// TIA Portal V17 export
// export: Created 2023-02-14T02:49:46.84947Z, ExportSetting WithDefaults, DisplayName Totally Integrated Automation Portal, DisplayVersion V17, DisplayName TIA Portal Openness, DisplayVersion V17, DisplayName TIA Portal Teamcenter Gateway, DisplayVersion V17, DisplayName TIA Portal Version Control Interface, DisplayVersion V17, DisplayName SINAMICS Startdrive Advanced, DisplayVersion V17, DisplayName SINAMICS Startdrive G130, G150, S120, S150, SINAMICS MV, S210, DisplayVersion V17, DisplayName SINAMICS Startdrive G110M, G120, G120C, G120D, G120P, G115D, DisplayVersion V17, DisplayName STEP 7 Professional, DisplayVersion V17, DisplayName STEP 7 Safety, DisplayVersion V17, DisplayName WinCC Professional, DisplayVersion V17
DATA_BLOCK "T-13.00_Homomixer"   // DB103
VERSION : 0.1
// stored: AutoNumber false, DBAccessibleFromOPCUA true, DBAccessibleFromWebserver true, InstanceOfName Homomix, InstanceOfType FB
"Homomix"
   // VAR_INPUT
   //    "Level LL" : Bool;
   //    IN_FBAV_ProWater : Bool;
   //    IN_FBAV_HW : Bool;
   //    IN_FBAV_CIP_Tank : Bool;
   //    IN_FBAV_CIP_Line : Bool;
   //    IN_FBAV_Outlet : Bool;
   //    IN_FBAV_Transfer : Bool;
   //    IN_FBP_Transfer : Bool;
   //    IN_FBP_Transfer_SP : Real;
   //    IN_FBP_CIP : Bool;
   //    IN_FBP_CIP_SP : Real;
   //    IN_CIP_Enable : Bool;
   //    IN_CIP_LineOpen : Bool;
   //    "CIP Pulse" : Bool;
   //    "CIP Request OK" : Bool;
   //    "CIP Supply ON" : Bool;
   //    "CIP In Progress" : Bool;
   //    "CIP Complete" : Bool;
   //    IN_Dose_Run : Bool;
   //    IN_Dose_Held : Bool;
   //    IN_Dose_Complete : Bool;
   //    IN_Dose_Valve_Cmd : Bool;
   //    IN_Dose_Pump_Cmd : Bool;
   //    IN_Dose_Pump_Sp : Real;
   //    IN_Dose_LineOK : Bool;
   //    "ProWater Ready" : Bool;
   //    "ProWater En" : Bool;
   //    "HW Ready" : Bool;
   //    "HW En" : Bool;
   //    "CIP Busy" : Bool;
   //    IN_LDT : Date_And_Time;
   // END_VAR
   // VAR_OUTPUT
   //    Out_AV_ProWater : Bool;
   //    Out_AV_HW : Bool;
   //    Out_AV_CIP_Tank : Bool;
   //    Out_AV_CIP_Line : Bool;
   //    Out_AV_Outlet : Bool;
   //    Out_AV_Transfer : Bool;
   //    Out_P_Transfer : Bool;
   //    Out_P_Transfer_SP : Real;
   //    Out_P_CIP : Bool;
   //    Out_P_CIP_SP : Real;
   //    Out_XA : Bool;
   //    Out_XA_SP : Real;
   //    Out_Prod_Ready : Bool;
   //    Out_Tank_Ready : Bool;
   //    Out_CIP_Tank_Req : Bool;
   //    Out_CIP_Line_Req : Bool;
   //    Out_CIP_LineOpen : Bool;
   // END_VAR
   // VAR
   //    Cmd : Struct
   //       Ready_for_Transfer : Bool;
   //       "CIP Tank" : Bool;
   //       "CIP Line" : Bool;
   //       "Agi Mode" : Bool;
   //       "Agi ON OFF" : Bool;
   //    END_STRUCT;
   // END_VAR
   // VAR RETAIN
   //    Param : Struct
   //       "CIP Pump SP" : Real;
   //       "Agi SP" : Real;
   //       Dose_HW_SP : Real;
   //       Dose_ProWater_SP : Real;
   //       LastDose_HW : Real;
   //       LastDose_ProWater : Real;
   //    END_STRUCT;
   // END_VAR
   // VAR
   //    State : Struct
   //       "Tank LL" : Bool;
   //       "CIP Tank" : Bool;
   //       "CIP Tank Ena" : Bool;
   //       "CIP Line" : Bool;
   //       "CIP Line Ena" : Bool;
   //       "CIP Return On" : Bool;
   //       "Dose EN" : Bool;
   //       ProWater_Inloading : Bool;
   //       HW_Inloading : Bool;
   //       Tank_Inloading : Bool;
   //       "Ready For Transfer" : Bool;
   //       "Ready For Transfer EN" : Bool;
   //       Transfer_On_Prog : Bool;
   //       "CIP Req" : Bool;
   //    END_STRUCT;
   //    Dose : Struct
   //       Dose_Start : DWord;
   //       Dose_Pause : DWord;
   //       Dose_Stop : DWord;
   //       Dose_State : DWord;
   //       Dose_Tank_Available : Word;
   //       Dose_Prod_Ready : Word;
   //       Dose_Header_Req : DWord;
   //       Dose_EN : Word;
   //    END_STRUCT;
   //    SP_ProWater : "Raw_Pulse";
   //    SP_HW { S7_SetPoint := 'True'} : "Raw_Pulse";
   //    Dose_ProWater { S7_SetPoint := 'True'} : "DOSE";
   //    Dose_HW { S7_SetPoint := 'True'} : "DOSE";
   //    r : Struct
   //       PosE1 : Bool;
   //       PosE2 : Bool;
   //       PosE3 : Bool;
   //       PosE4 : Bool;
   //       PosE5 : Bool;
   //       PosE6 : Bool;
   //       PosE7 : Bool;
   //       PosE8 : Bool;
   //       PosE9 : Bool;
   //       PosE10 : Bool;
   //       PosE11 : Bool;
   //       PosE12 : Bool;
   //       PosE13 : Bool;
   //       PosE14 : Bool;
   //       PosE15 : Bool;
   //       PosE16 : Bool;
   //       PosE17 : Bool;
   //       PosE18 : Bool;
   //       PosE19 : Bool;
   //       PosE20 : Bool;
   //       PosE21 : Bool;
   //       PosE22 : Bool;
   //       PosE23 : Bool;
   //       PosE24 : Bool;
   //       PosE25 : Bool;
   //       PosE26 : Bool;
   //       PosE27 : Bool;
   //       PosE28 : Bool;
   //       PosE29 : Bool;
   //       PosE30 : Bool;
   //       PosE31 : Bool;
   //       PosE32 : Bool;
   //    END_STRUCT;
   //    CIPRetOn_Time : TON_TIME;
   //    CIPRetOff_Time { S7_SetPoint := 'True'} : TON_TIME;
   //    Actuator : Struct
   //       AV_Transfer : Bool;
   //       AV_Outlet : Bool;
   //       AV_CIP : Bool;
   //       P_Transfer : Bool;
   //       P_CIP : Bool;
   //    END_STRUCT;
   //    alwaysOn : Bool;
   // END_VAR
   // VAR RETAIN
   //    TimerON : Struct
   //       TimerON_1 : TON_TIME;
   //       TimerON_2 { S7_SetPoint := 'True'} : TON_TIME;
   //       TimerON_3 { S7_SetPoint := 'True'} : TON_TIME;
   //       TimerON_4 { S7_SetPoint := 'True'} : TON_TIME;
   //       TimerON_5 { S7_SetPoint := 'True'} : TON_TIME;
   //       TimerON_6 { S7_SetPoint := 'True'} : TON_TIME;
   //       TimerON_7 { S7_SetPoint := 'True'} : TON_TIME;
   //       TimerON_8 { S7_SetPoint := 'True'} : TON_TIME;
   //    END_STRUCT;
   // END_VAR
BEGIN
END_DATA_BLOCK
